// TwinCAT 3 PLC project Untitled1
// ProgramVersion: 3.1.4023.0
// libraries:
//   Tc2_Standard, * (Beckhoff Automation GmbH)
//   Tc2_System, * (Beckhoff Automation GmbH)
//   Tc3_Module, * (Beckhoff Automation GmbH)
// project tree:
//   / PlcTask.TcTTO
//   POUs/ FB_TwinCat.TcPOU, MAIN.TcPOU
// real-time tasks:
//   TASK PlcTask: cycle T#10ms, priority 20, ADS port 350

CONFIGURATION Untitled1
    RESOURCE PLC ON TwinCAT3
        TASK PlcTask(INTERVAL := T#10ms, PRIORITY := 20);
        PROGRAM MAIN WITH PlcTask : MAIN;
    END_RESOURCE
END_CONFIGURATION

// ---- POUs/MAIN.TcPOU
PROGRAM MAIN
VAR
END_VAR

END_PROGRAM

// ---- POUs/FB_TwinCat.TcPOU
FUNCTION_BLOCK FB_TwinCat
VAR_INPUT
	input	:	BOOL;
	inputreal:	REAL;
END_VAR
VAR_OUTPUT
	outputreal			:	real;
END_VAR
VAR
END_VAR

IF input=TRUE THEN
	outputreal:=inputreal;
END_IF
//oder
IF 			input=FALSE THEN
	outputreal:=inputreal/2;
END_IF;

END_FUNCTION_BLOCK
